FUNCTION_BLOCK SDInitDone (* Basic Function Block Type *)
  (* Standard: 61499-2 *)
  (* Version 0.0, 7/30/2026, Schneider Electric, Template *)
  PACKAGE SE.Nereda;
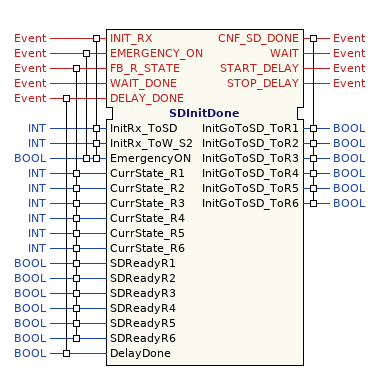
  EVENT_INPUT
    INIT_RX WITH InitRx_ToSD, InitRx_ToW_S2, EmergencyON; (* Initialization Request *)
    EMERGENCY_ON WITH EmergencyON;
    FB_R_STATE WITH CurrState_R1, CurrState_R2, CurrState_R3, CurrState_R4, CurrState_R5, CurrState_R6, SDReadyR1, SDReadyR2, SDReadyR3, SDReadyR4, SDReadyR5, SDReadyR6;
    WAIT_DONE;
    DELAY_DONE WITH DelayDone;
  END_EVENT
  EVENT_OUTPUT
    CNF_SD_DONE WITH InitGoToSD_ToR1, InitGoToSD_ToR2, InitGoToSD_ToR3, InitGoToSD_ToR4, InitGoToSD_ToR5, InitGoToSD_ToR6; (* Execution Confirmation *)
    WAIT;
    START_DELAY;
    STOP_DELAY;
  END_EVENT
  VAR_INPUT
    InitRx_ToSD : INT; (* Input event qualifier *)
    InitRx_ToW_S2 : INT;
    EmergencyON : BOOL;
    CurrState_R1 : INT;
    CurrState_R2 : INT;
    CurrState_R3 : INT;
    CurrState_R4 : INT;
    CurrState_R5 : INT;
    CurrState_R6 : INT;
    SDReadyR1 : BOOL;
    SDReadyR2 : BOOL;
    SDReadyR3 : BOOL;
    SDReadyR4 : BOOL;
    SDReadyR5 : BOOL;
    SDReadyR6 : BOOL;
    DelayDone : BOOL;
  END_VAR
  VAR_OUTPUT
    InitGoToSD_ToR1 : BOOL; (* Output event qualifier *)
    InitGoToSD_ToR2 : BOOL;
    InitGoToSD_ToR3 : BOOL;
    InitGoToSD_ToR4 : BOOL;
    InitGoToSD_ToR5 : BOOL;
    InitGoToSD_ToR6 : BOOL;
  END_VAR
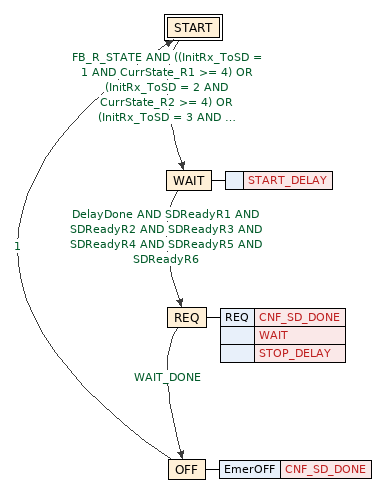
  EC_STATES
    START; (* Initial State *)
    REQ : REQ -> CNF_SD_DONE, -> WAIT, -> STOP_DELAY;
    OFF : EmerOFF -> CNF_SD_DONE;
    WAIT : -> START_DELAY;
  END_STATES
  EC_TRANSITIONS
    START TO WAIT := FB_R_STATE AND ((InitRx_ToSD = 1 AND CurrState_R1 >= 4) OR (InitRx_ToSD = 2 AND CurrState_R2 >= 4) OR (InitRx_ToSD = 3 AND CurrState_R3 >= 4) OR (InitRx_ToSD = 4 AND CurrState_R4 >= 4) OR (InitRx_ToSD = 5 AND CurrState_R5 >= 4) OR (InitRx_ToSD = 6 AND CurrState_R6 >= 4));
    REQ TO OFF := WAIT_DONE;
    OFF TO START := 1;
    WAIT TO REQ := DelayDone AND SDReadyR1 AND SDReadyR2 AND SDReadyR3 AND SDReadyR4 AND SDReadyR5 AND SDReadyR6;
  END_TRANSITIONS
  ALGORITHM REQ IN ST: (* Normally executed algorithm *)
;
IF InitRx_ToW_S2 = 1 THEN
	InitGoToSD_ToR1 := TRUE;

ELSIF InitRx_ToW_S2 = 2 THEN
	InitGoToSD_ToR2 := TRUE;

ELSIF InitRx_ToW_S2 = 3 THEN
	InitGoToSD_ToR3 := TRUE;

ELSIF InitRx_ToW_S2 = 4 THEN
	InitGoToSD_ToR4 := TRUE;

ELSIF InitRx_ToW_S2 = 5 THEN
	InitGoToSD_ToR5 := TRUE;

ELSIF InitRx_ToW_S2 = 6 THEN
	InitGoToSD_ToR6 := TRUE;
END_IF;
  END_ALGORITHM
  ALGORITHM EmerOFF IN ST:
;
InitGoToSD_ToR1 := FALSE;
InitGoToSD_ToR2 := FALSE;
InitGoToSD_ToR3 := FALSE;
InitGoToSD_ToR4 := FALSE;
InitGoToSD_ToR5 := FALSE;
InitGoToSD_ToR6 := FALSE;
  END_ALGORITHM
END_FUNCTION_BLOCK
